PROGRAM MAIN_1
VAR
END_VAR


Camera();

END_PROGRAM

(* stored: Version 1.1.0.1, ProductVersion 3.1.4024.12
   POU MAIN_1: Id {e1836af3-81b1-400d-b275-7e28fbb3edc4}, SpecialFunc None *)
